FUNCTION_BLOCK FB_S_Temperatursensor IMPLEMENTS	I_Sensor	
VAR_INPUT
	I_iSignal			:INT;		// Messsignal des Sensors
	I_rHigh				:REAL;		// Oberer Schwellenwert für Prozess
	I_rLow				:REAL;		// Unterer Schwellenwert für Prozess
	I_rMax				:REAL;		// Skallierungswert -> Max-Wert 
	I_rMin				:REAL;		// Skallierungswert -> Min-Wert 
END_VAR

VAR_OUTPUT
	O_bStoerung			:BOOL;		// Befindet sich das Element in einem Error
	O_iStoerungID		:INT;		// Anzeigen von Störung über eine INT-Variable
END_VAR

VAR
	Messwert			:REAL;		// Wert für HMI
	GrenzeOben			:BOOL;		// Wert für HMI
	GrenzeUnten			:BOOL;		// Wert für HMI
END_VAR

Messwert := P_Messwert;
GrenzeOben := P_GrenzeOben;
GrenzeUnten := P_GrenzeUnten;

PROPERTY PUBLIC P_GrenzeOben : BOOL
GET
IF P_Messwert > I_rHigh THEN
	P_GrenzeOben := TRUE;
ELSE
	P_GrenzeOben := FALSE;
END_IF
END_GET
END_PROPERTY

PROPERTY PUBLIC P_GrenzeUnten : BOOL
GET
IF P_Messwert < I_rLow THEN
	P_GrenzeUnten := TRUE;
ELSE
	P_GrenzeUnten := FALSE;
END_IF
END_GET
END_PROPERTY

PROPERTY PUBLIC P_Messwert : REAL
GET
IF I_iSignal > 27648 OR I_iSignal < 0 THEN
	O_bStoerung := TRUE;
	O_iStoerungID := 04;
ELSE
	O_bStoerung := FALSE; 
END_IF

// Linearisierung des Wertes 
P_Messwert := INT_TO_REAL(I_iSignal) * (I_rMax-I_rMin) / 27648 + I_rMin;
END_GET
END_PROPERTY

END_FUNCTION_BLOCK

(* stored: Version 1.1.0.1, ProductVersion 3.1.4024.12
   POU FB_S_Temperatursensor: Id {fbd32386-a253-49ea-826a-bfbe4aab9dab}, SpecialFunc None
   Property P_GrenzeOben: Id {e3d174c2-5619-46cb-b6e5-a2971410ae38}
   Get Get: Id {c1944f02-f458-40d4-9cce-8887d1cab55d}
   Property P_GrenzeUnten: Id {8b7656b1-9197-4364-a830-ee1874b698bf}
   Get Get: Id {055193c3-c26f-4f59-a9f9-fe3fe7d25c0d}
   Property P_Messwert: Id {bd948508-785d-4a27-9dd5-c30f6507186a}
   Get Get: Id {d9634401-2e84-4702-b005-564f875f3833} *)
